// TIA Portal V17 export
// export: Created 2025-03-07T09:19:39.3873265Z, ExportSetting WithDefaults, DisplayName Totally Integrated Automation Portal, DisplayVersion V17 Update 8, DisplayName TIA Portal Openness, DisplayVersion V17 Update 8, DisplayName TIA Portal Version Control Interface, DisplayVersion V17, DisplayName SINAMICS Startdrive Advanced, DisplayVersion V17 SP2, DisplayName SINAMICS Startdrive G110M, G120, G120C, G120D, G120P, G115D, DisplayVersion V17 SP2, DisplayName SINAMICS Startdrive G130, G150, S120, S150, SINAMICS MV, S210, DisplayVersion V17 SP2, DisplayName STEP 7 Professional, DisplayVersion V17 Update 8, DisplayName SINUMERIK ONE STEP 7 Toolbox, DisplayVersion V17 Update 12, DisplayName SINUMERIK 840D sl STEP 7 Toolbox, DisplayVersion V17 Update 12, DisplayName STEP 7 Safety, DisplayVersion V17 Update 6, DisplayName WinCC Advanced, DisplayVersion V17 Update 8
TYPE "READ_TOOL_DATA_SP1"
// stored: IsFailsafeCompliant false
   STRUCT
      READ : Struct
         FB2_DATA_SP1 : Struct
            Error : Bool;   // Error
            Done : Bool;   // Done
            Request : Bool;   // Request
            Error_Fault : Bool;   // Error Fault
            Status : Word;   // Pulse
            MAG_POS_IN_NC : Int;   // MAGAZINE POSITION IN NC
            Tool_state : Word;   // Tool state
            TOOL_NUMBER : Int;   // TOOL NUMBER
            MAGAZINE_POSITION : Int;   // MAGAZINE POSITION
         END_STRUCT;
         TOOL_DATA_SP1 : Struct   // TOOL DATA
            NUM_CUTING_EDGE : Int;   // NUM CUTING EDGE
            QUANTITY_EDGE : Array[1..5] of Real;   // QUANTITY EDGE
            WARNING_EDGE : Array[1..5] of Real;   // WARNING EDGE
            EXPIRED_EDGE : Array[1..5] of Real;   // EXPIRED EDGE
         END_STRUCT;
         PARAM_SPINDLE_SP1 : Struct
            TC_MOP4_QUANTITY_1 : Struct
               SYNTAX_ID : Byte := BYTE#16#82;   // SYNTAX ID
               AREA_UNIT : Byte := BYTE#16#81;   // AREA UNIT
               COLUMN : Word := 16#0;   // TOOL NUMBER (HEX)
               LINE : Word := WORD#16#0004;   // $TC_MOP4[TOOL,1] CUTTING REMAINING LIFE COUNTER
               BLOCKTYPE : Byte := BYTE#16#22;   // BLOCKTYPE
               NUMOFLINE : Byte := BYTE#16#01;   // NUMOFLINE
               DATATYPE : Byte := BYTE#16#0F;   // DATATYPE
               LENGTH : Byte := BYTE#16#08;   // LENGTH
            END_STRUCT;
            TC_MOP4_QUANTITY_2 : Struct
               SYNTAX_ID : Byte := BYTE#16#82;
               AREA_UNIT : Byte := BYTE#16#81;
               COLUMN : Word := 16#0;   // TOOL NUMBER (HEX)
               LINE : Word := WORD#16#000D;   // $TC_MOP4[TOOL,2] CUTTING REMAINING LIFE COUNTER
               BLOCKTYPE : Byte := BYTE#16#22;
               NUMOFLINE : Byte := BYTE#16#01;
               DATATYPE : Byte := BYTE#16#0F;
               LENGTH : Byte := BYTE#16#08;
            END_STRUCT;
            TC_MOP4_QUANTITY_3 : Struct
               SYNTAX_ID : Byte := BYTE#16#82;
               AREA_UNIT : Byte := BYTE#16#81;
               COLUMN : Word := 16#0;   // TOOL NUMBER (HEX)
               LINE : Word := WORD#16#0016;   // $TC_MOP4[TOOL,3] CUTTING REMAINING LIFE COUNTER
               BLOCKTYPE : Byte := BYTE#16#22;
               NUMOFLINE : Byte := BYTE#16#01;
               DATATYPE : Byte := BYTE#16#0F;
               LENGTH : Byte := BYTE#16#08;
            END_STRUCT;
            TC_MOP4_QUANTITY_4 : Struct
               SYNTAX_ID : Byte := BYTE#16#82;
               AREA_UNIT : Byte := BYTE#16#81;
               COLUMN : Word := 16#0;   // TOOL NUMBER (HEX)
               LINE : Word := WORD#16#001F;   // $TC_MOP4[TOOL,4] CUTTING REMAINING LIFE COUNTER
               BLOCKTYPE : Byte := BYTE#16#22;
               NUMOFLINE : Byte := BYTE#16#01;
               DATATYPE : Byte := BYTE#16#0F;
               LENGTH : Byte := BYTE#16#08;
            END_STRUCT;
            TC_MOP4_QUANTITY_5 : Struct
               SYNTAX_ID : Byte := BYTE#16#82;
               AREA_UNIT : Byte := BYTE#16#81;
               COLUMN : Word := 16#0;   // TOOL NUMBER (HEX)
               LINE : Word := WORD#16#0028;   // $TC_MOP4[TOOL,4] CUTTING REMAINING LIFE COUNTER / $TC_MOP4[TOOL,5] CUTTING REMAINING LIFE COUNTER
               BLOCKTYPE : Byte := BYTE#16#22;
               NUMOFLINE : Byte := BYTE#16#01;
               DATATYPE : Byte := BYTE#16#0F;
               LENGTH : Byte := BYTE#16#08;
            END_STRUCT;
            TC_MOP3_WARNING_1 : Struct
               SYNTAX_ID : Byte := BYTE#16#82;
               AREA_UNIT : Byte := BYTE#16#81;
               COLUMN : Word := 16#0;   // TOOL NUMBER (HEX)
               LINE : Word := WORD#16#0003;   // $TC_MOP3[TOOL,1] CUTTING PREWARNING LIFE COUNTER
               BLOCKTYPE : Byte := BYTE#16#22;
               NUMOFLINE : Byte := BYTE#16#01;
               DATATYPE : Byte := BYTE#16#0F;
               LENGTH : Byte := BYTE#16#08;
            END_STRUCT;
            TC_MOP3_WARNING_2 : Struct
               SYNTAX_ID : Byte := BYTE#16#82;
               AREA_UNIT : Byte := BYTE#16#81;
               COLUMN : Word := 16#0;   // TOOL NUMBER (HEX)
               LINE : Word := WORD#16#000C;   // $TC_MOP3[TOOL,2] CUTTING PREWARNING LIFE COUNTER
               BLOCKTYPE : Byte := BYTE#16#22;
               NUMOFLINE : Byte := BYTE#16#01;
               DATATYPE : Byte := BYTE#16#0F;
               LENGTH : Byte := BYTE#16#08;
            END_STRUCT;
            TC_MOP3_WARNING_3 : Struct
               SYNTAX_ID : Byte := BYTE#16#82;
               AREA_UNIT : Byte := BYTE#16#81;
               COLUMN : Word := 16#0;   // TOOL NUMBER (HEX)
               LINE : Word := WORD#16#0015;   // $TC_MOP3[TOOL,3] CUTTING PREWARNING LIFE COUNTER
               BLOCKTYPE : Byte := BYTE#16#22;
               NUMOFLINE : Byte := BYTE#16#01;
               DATATYPE : Byte := BYTE#16#0F;
               LENGTH : Byte := BYTE#16#08;
            END_STRUCT;
            TC_MOP3_WARNING_4 : Struct
               SYNTAX_ID : Byte := BYTE#16#82;
               AREA_UNIT : Byte := BYTE#16#81;
               COLUMN : Word := 16#0;   // TOOL NUMBER (HEX)
               LINE : Word := WORD#16#001E;   // $TC_MOP3[TOOL,4] CUTTING PREWARNING LIFE COUNTER
               BLOCKTYPE : Byte := BYTE#16#22;
               NUMOFLINE : Byte := BYTE#16#01;
               DATATYPE : Byte := BYTE#16#0F;
               LENGTH : Byte := BYTE#16#08;
            END_STRUCT;
            TC_MOP3_WARNING_5 : Struct
               SYNTAX_ID : Byte := BYTE#16#82;
               AREA_UNIT : Byte := BYTE#16#81;
               COLUMN : Word := 16#0;   // TOOL NUMBER (HEX)
               LINE : Word := WORD#16#0027;   // $TC_MOP3[TOOL,4] CUTTING PREWARNING LIFE COUNTER / $TC_MOP3[TOOL,5] CUTTING PREWARNING LIFE COUNTER
               BLOCKTYPE : Byte := BYTE#16#22;
               NUMOFLINE : Byte := BYTE#16#01;
               DATATYPE : Byte := BYTE#16#0F;
               LENGTH : Byte := BYTE#16#08;
            END_STRUCT;
            TC_MOP13_EXPIRED_1 : Struct
               SYNTAX_ID : Byte := BYTE#16#82;
               AREA_UNIT : Byte := BYTE#16#81;
               COLUMN : Word := 16#0;   // TOOL NUMBER (HEX)
               LINE : Word := WORD#16#0006;   // $TC_MOP13[TOOL,1] CUTTING SET POINT LIFE COUNTER
               BLOCKTYPE : Byte := BYTE#16#22;
               NUMOFLINE : Byte := BYTE#16#01;
               DATATYPE : Byte := BYTE#16#0F;
               LENGTH : Byte := BYTE#16#08;
            END_STRUCT;
            TC_MOP13_EXPIRED_2 : Struct
               SYNTAX_ID : Byte := BYTE#16#82;
               AREA_UNIT : Byte := BYTE#16#81;
               COLUMN : Word := 16#0;   // TOOL NUMBER (HEX)
               LINE : Word := WORD#16#000F;   // $TC_MOP13[TOOL,2] CUTTING SET POINT LIFE COUNTER
               BLOCKTYPE : Byte := BYTE#16#22;
               NUMOFLINE : Byte := BYTE#16#01;
               DATATYPE : Byte := BYTE#16#0F;
               LENGTH : Byte := BYTE#16#08;
            END_STRUCT;
            TC_MOP13_EXPIRED_3 : Struct
               SYNTAX_ID : Byte := BYTE#16#82;
               AREA_UNIT : Byte := BYTE#16#81;
               COLUMN : Word := 16#0;   // TOOL NUMBER (HEX)
               LINE : Word := WORD#16#0018;   // $TC_MOP13[TOOL,3] CUTTING SET POINT LIFE COUNTER
               BLOCKTYPE : Byte := BYTE#16#22;
               NUMOFLINE : Byte := BYTE#16#01;
               DATATYPE : Byte := BYTE#16#0F;
               LENGTH : Byte := BYTE#16#08;
            END_STRUCT;
            TC_MOP13_EXPIRED_4 : Struct
               SYNTAX_ID : Byte := BYTE#16#82;
               AREA_UNIT : Byte := BYTE#16#81;
               COLUMN : Word := 16#0;   // TOOL NUMBER (HEX)
               LINE : Word := WORD#16#0021;   // $TC_MOP13[TOOL,4] CUTTING SET POINT LIFE COUNTER
               BLOCKTYPE : Byte := BYTE#16#22;
               NUMOFLINE : Byte := BYTE#16#01;
               DATATYPE : Byte := BYTE#16#0F;
               LENGTH : Byte := BYTE#16#08;
            END_STRUCT;
            TC_MOP13_EXPIRED_5 : Struct
               SYNTAX_ID : Byte := BYTE#16#82;
               AREA_UNIT : Byte := BYTE#16#81;
               COLUMN : Word := 16#0;   // TOOL NUMBER (HEX)
               LINE : Word := WORD#16#002A;   // $TC_MOP13[TOOL,4] CUTTING SET POINT LIFE COUNTER / $TC_MOP13[TOOL,5] CUTTING SET POINT LIFE COUNTER
               BLOCKTYPE : Byte := BYTE#16#22;
               NUMOFLINE : Byte := BYTE#16#01;
               DATATYPE : Byte := BYTE#16#0F;
               LENGTH : Byte := BYTE#16#08;
            END_STRUCT;
         END_STRUCT;
         FB2_VARS_SP1 : Struct
            TOOL_NUMBER : Struct
               error : Bool;
               done : Bool;
               request : Bool;
            END_STRUCT;
            ORIGI_MAGAZINE : Struct
               error : Bool;
               done : Bool;
               request : Bool;
            END_STRUCT;
            CUTING_EDGE : Struct
               error : Bool;
               done : Bool;
               request : Bool;
            END_STRUCT;
            QUANTITY_EDGE : Struct
               error : Bool;
               done : Bool;
               request : Bool;
            END_STRUCT;
            WARNING_EDGE : Struct
               error : Bool;
               done : Bool;
               request : Bool;
            END_STRUCT;
            EXPIRED_EDGE : Struct
               error : Bool;
               done : Bool;
               request : Bool;
            END_STRUCT;
         END_STRUCT;
         SMNS_PRMTRS_SP1 : Struct
            TC_MPP6_PLACE_DATA : Struct
               SYNTAX_ID : Byte := BYTE#16#82;
               AREA_UNIT : Byte := BYTE#16#81;   // CHANNEL NUMBER, 81=CH1, 82=CH2 )
               COLUMN : Word := WORD#16#0001;   // MAGAZINE NUMBER
               LINE : Word := 16#0;
               BLOCKTYPE : Byte := BYTE#16#28;
               NUMOFLINE : Byte := BYTE#16#01;
               DATATYPE : Byte := BYTE#16#04;
               LENGTH : Byte := BYTE#16#02;
            END_STRUCT;
            NUM_CUTTING_EDGES : Struct
               SYNTAX_ID : Byte := BYTE#16#82;
               AREA_UNIT : Byte := BYTE#16#81;
               COLUMN : Word := WORD#16#000E;   // NUM CUTTING EDGES
               LINE : Word := WORD#16#0001;
               BLOCKTYPE : Byte := BYTE#16#21;
               NUMOFLINE : Byte := BYTE#16#01;
               DATATYPE : Byte := BYTE#16#04;
               LENGTH : Byte := BYTE#16#02;
            END_STRUCT;
            DUPLO_NUMBER : Struct
               SYNTAX_ID : Byte := BYTE#16#82;
               AREA_UNIT : Byte := BYTE#16#81;
               COLUMN : Word := WORD#16#0002;   // DUPLO NUMBER
               LINE : Word := WORD#16#0001;
               BLOCKTYPE : Byte := BYTE#16#21;
               NUMOFLINE : Byte := BYTE#16#01;
               DATATYPE : Byte := BYTE#16#04;
               LENGTH : Byte := BYTE#16#02;
            END_STRUCT;
            ORIG_MAGAZINE : Struct
               SYNTAX_ID : Byte := BYTE#16#82;
               AREA_UNIT : Byte := BYTE#16#81;
               COLUMN : Word := WORD#16#0011;   // ORIG MAGAZINE
               LINE : Word := WORD#16#0001;
               BLOCKTYPE : Byte := BYTE#16#21;
               NUMOFLINE : Byte := BYTE#16#01;
               DATATYPE : Byte := BYTE#16#04;
               LENGTH : Byte := BYTE#16#02;
            END_STRUCT;
         END_STRUCT;
      END_STRUCT;
   END_STRUCT;
   // // READ.TOOL_DATA_SP1.QUANTITY_EDGE[1] : QUANTITY EDGE[1]
   // // READ.TOOL_DATA_SP1.QUANTITY_EDGE[2] : QUANTITY EDGE[2]
   // // READ.TOOL_DATA_SP1.QUANTITY_EDGE[3] : QUANTITY EDGE[3]
   // // READ.TOOL_DATA_SP1.QUANTITY_EDGE[4] : QUANTITY EDGE[4]
   // // READ.TOOL_DATA_SP1.QUANTITY_EDGE[5] : QUANTITY EDGE[5]
   // // READ.TOOL_DATA_SP1.WARNING_EDGE[1] : WARNING EDGE[1]
   // // READ.TOOL_DATA_SP1.WARNING_EDGE[2] : WARNING EDGE[2]
   // // READ.TOOL_DATA_SP1.WARNING_EDGE[3] : WARNING EDGE[3]
   // // READ.TOOL_DATA_SP1.WARNING_EDGE[4] : WARNING EDGE[4]
   // // READ.TOOL_DATA_SP1.WARNING_EDGE[5] : WARNING EDGE[5]
   // // READ.TOOL_DATA_SP1.EXPIRED_EDGE[1] : EXPIRED EDGE[1]
   // // READ.TOOL_DATA_SP1.EXPIRED_EDGE[2] : EXPIRED EDGE[2]
   // // READ.TOOL_DATA_SP1.EXPIRED_EDGE[3] : EXPIRED EDGE[3]
   // // READ.TOOL_DATA_SP1.EXPIRED_EDGE[4] : EXPIRED EDGE[4]
   // // READ.TOOL_DATA_SP1.EXPIRED_EDGE[5] : EXPIRED EDGE[5]
END_TYPE
